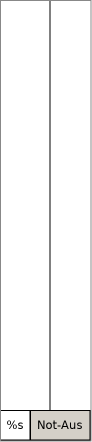
VISUALIZATION V_LiquidTransorState  // 92x442
VAR_IN_OUT
	IOfbTransor : FB_Transor;
END_VAR
    Rectangle (0,410 30x30), "%s", text variable: IOfbTransor.iChan
    Rectangle (30,410 60x30), "Not-Aus", colour toggle: IOfbTransor.QbTransor
    Line (50,410) (50,0), colour toggle: IOfbTransor.QbTransor
END_VISUALIZATION

(* stored: Version 1.1.0.1, ProductVersion 3.1.4018.10
   Visu V_LiquidTransorState: Id {c749067f-e4fd-46fd-9edb-2d6372d0c0bc} *)
